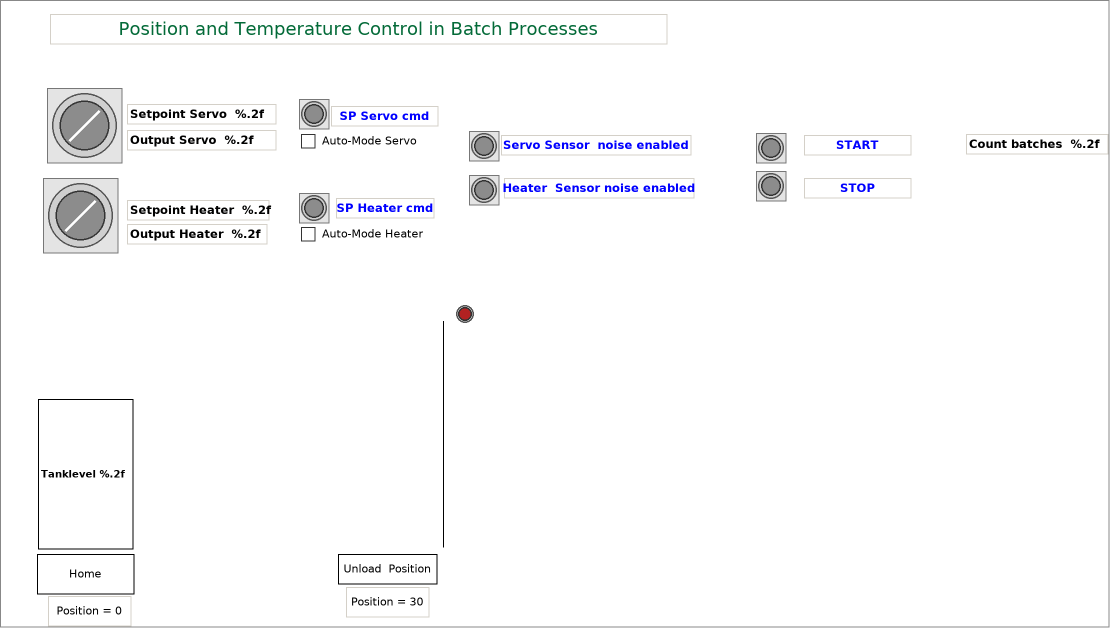
VISUALIZATION UserInterface  // 1110x628
    PushSwitch (299,99 30x30), variable: GVL_IO.xPushButton1, behaviour: TAP, style: Switch-PushSwitch-Gray
    Potentiometer360 (47,88 75x75), variable: GVL_IO.SetPoint_ServoX, style: Potentiometer-Potentiometer360-Gray, scale format: %d, scale 0..60
        p2431819421: Outside
    Textfield (127,104 149x20), "Setpoint Servo %.2f", text variable: GVL_IO.SetPoint_ServoX
    Textfield (127,130 149x20), "Output Servo %.2f", text variable: GVL_IO.Output_ServoX
    Potentiometer360 (43,178 75x75), variable: GVL_IO.SetPointHeater, style: Potentiometer-Potentiometer360-Gray, scale format: %d, scale 15..115
        p2431819421: Outside
    PushSwitch (299,193 30x30), variable: GVL_IO.xPushButton2, behaviour: TAP, style: Switch-PushSwitch-Gray
    Textfield (127,200 142x20), "Setpoint Heater %.2f", text variable: GVL_IO.SetPointHeater
    Textfield (127,224 140x20), "Output Heater %.2f", text variable: GVL_IO.Output_Heater
    Rectangle (37,554 97x40), "Home"
    Rectangle (338,554 99x30), "Unload Position"
    Textfield (346,587 83x30), "Position = 30"
    Textfield (48,596 83x30), "Position = 0"
    Rectangle (38,399 95x150), "Tanklevel %.2f", text variable: GVL_IO.TankLevelSensor
        p3560616238: GVL_IO.Output_ServoX * 10
    Textfield (336,198 98x20), "SP Heater cmd"
    Textfield (331,106 107x20), "SP Servo cmd"
    Textfield (50,14 617x30), "Position and Temperature Control in Batch Processes"
    Checkbox (299,224 125x20), "Auto-Mode Heater", variable: MAIN.PIDheater_on
    Checkbox (299,131 195x20), "Auto-Mode Servo", variable: MAIN.PIDServo_on
    Line (443,321) (443,547)
    Lamp1 (455,304 20x20), variable: (GVL_IO.Output_ServoX>31), style: Lamp-Lamp1-Red
    PushSwitch (469,175 30x30), variable: GVL_IO.noise_HeaterSensor, behaviour: TOGGLE, style: Switch-PushSwitch-Gray
    Textfield (504,178 190x20), "Heater Sensor noise enabled"
    PushSwitch (469,131 30x30), variable: GVL_IO.noise_ServoSensor, behaviour: TOGGLE, style: Switch-PushSwitch-Gray
    Textfield (501,135 190x20), "Servo Sensor noise enabled"
    PushSwitch (756,133 30x30), variable: GVL_IO.StartPr, behaviour: TOGGLE, style: Switch-PushSwitch-Gray
    PushSwitch (756,171 30x30), variable: GVL_IO.StopPr, behaviour: TOGGLE, style: Switch-PushSwitch-Gray
    Textfield (804,135 107x20), "START"
    Textfield (804,178 107x20), "STOP"
    Textfield (966,134 142x20), "Count batches %.2f", text variable: GVL_IO.countBatches
END_VISUALIZATION

(* stored: Version 1.1.0.1, ProductVersion 3.1.4024.2
   Visu UserInterface: Id {8126f8ab-e6ef-48b6-9ba2-149e11247293} *)
